// SIMATIC STEP 7 (V5.x) project Y_A start
// CPU: CPU 315
// station: Hardware
// station: SIMATIC 300(1)
// station: P_ADR_BUS
// program: S7 Program(3)

SYMBOL_TABLE
"Y_A"	FC 1	FC 1	// 星_三角 启动
"open"	I 0.0	BOOL	// 启动按钮
"stop"	I 0.1	BOOL	// 停止按钮
"over"	I 0.2	BOOL	// 过载保护
"T_km"	Q 4.0	BOOL	// 总接触器
"Y_km"	Q 4.1	BOOL	// 星点接触器
"A_km"	Q 4.2	BOOL	// 三角形接触器
"lamp"	Q 5.0	BOOL	// 运行指示灯
"timer0"	T 0	TIMER	// 星接延时
"timer1"	T 1	TIMER	// 断星接延时
"timer2"	T 2	TIMER	// 接通三角延时
END_SYMBOL_TABLE

FUNCTION "Y_A" : VOID	// FC 1
TITLE = 星_三角 启动电路
//这里星_三角 启动电路的功能模块。按启动按钮open后，运行指示lamp有指示，接触器T_km
//和Y_km接通，进行星形启动，时间为t0，然后断开T_km和Y_km，时间为t1，再接通A_km，延
//时t2时间后，再接通T_km，星三角启动完成。按停止按钮stop，或电路过载over，可停止电
//路运行。
VERSION : 0.1
VAR_INPUT
  open : BOOL ;	//启动按钮
  stop : BOOL ;	//停止按钮
  over : BOOL ;	//过载保护
  t0 : S5TIME ;	//星接延时时间
  t1 : S5TIME ;	//断开星接时间
  t2 : S5TIME ;	//接通三角时间
  timer0 : TIMER ;	//星接延时器
  timer1 : TIMER ;	//断星延时器
  timer2 : TIMER ;	//接角延时器
END_VAR
VAR_OUTPUT
  T_km : BOOL ;	//总接触器
  Y_km : BOOL ;	//星点接触器
  A_km : BOOL ;	//三角接触器
  lamp : BOOL ;	//运行指示
END_VAR
BEGIN
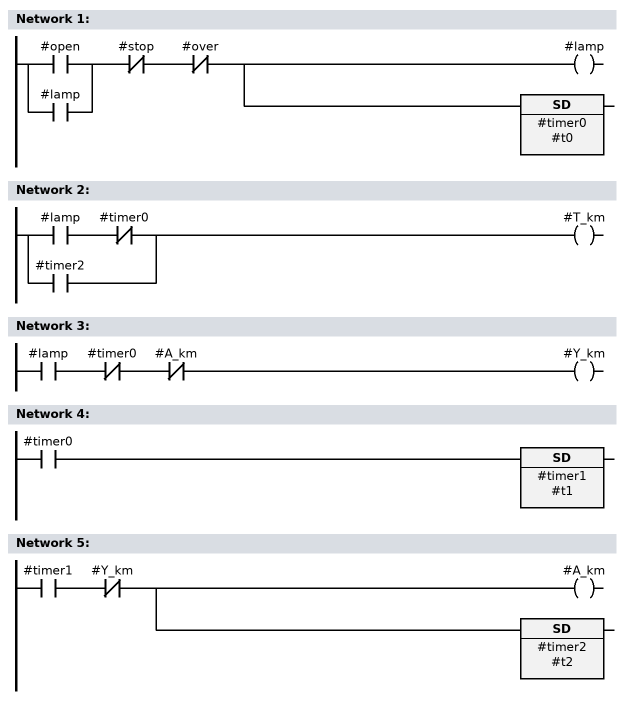
NETWORK
TITLE =
      A(;
      O     #open;
      O     #lamp;
      );
      AN    #stop;
      AN    #over;
      =     #lamp;
      L     #t0;
      SD    #timer0;
NETWORK
TITLE =
      A     #lamp;
      AN    #timer0;
      O     #timer2;
      =     #T_km;
NETWORK
TITLE =
      A     #lamp;
      AN    #timer0;
      AN    #A_km;
      =     #Y_km;
NETWORK
TITLE =
      A     #timer0;
      L     #t1;
      SD    #timer1;
NETWORK
TITLE =
      A     #timer1;
      AN    #Y_km;
      =     #A_km;
      L     #t2;
      SD    #timer2;
END_FUNCTION

ORGANIZATION_BLOCK OB 1
TITLE = "Main Program Sweep (Cycle)"
VERSION : 0.1
VAR_TEMP
  OB1_EV_CLASS : BYTE ;	//Bits 0-3 = 1 (Coming event), Bits 4-7 = 1 (Event class 1)
  OB1_SCAN_1 : BYTE ;	//1 (Cold restart scan 1 of OB 1), 3 (Scan 2-n of OB 1)
  OB1_PRIORITY : BYTE ;	//Priority of OB Execution
  OB1_OB_NUMBR : BYTE ;	//1 (Organization block 1, OB1)
  OB1_RESERVED_1 : BYTE ;	//Reserved for system
  OB1_RESERVED_2 : BYTE ;	//Reserved for system
  OB1_PREV_CYCLE : INT ;	//Cycle time of previous OB1 scan (milliseconds)
  OB1_MIN_CYCLE : INT ;	//Minimum cycle time of OB1 (milliseconds)
  OB1_MAX_CYCLE : INT ;	//Maximum cycle time of OB1 (milliseconds)
  OB1_DATE_TIME : DATE_AND_TIME ;	//Date and time OB1 started
END_VAR
BEGIN
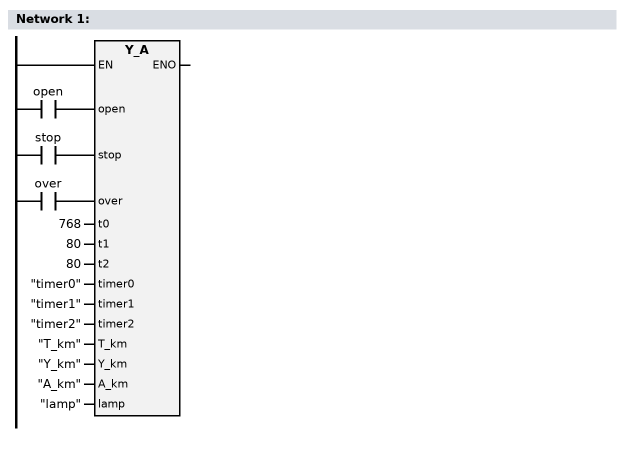
NETWORK
TITLE =
      A     "open";
      =     L 20.0;
      BLD   103;
      A     "stop";
      =     L 20.1;
      BLD   103;
      A     "over";
      =     L 20.2;
      BLD   103;
      CALL  "Y_A" (
           open                     := L 20.0,
           stop                     := L 20.1,
           over                     := L 20.2,
           t0                       := 768,
           t1                       := 80,
           t2                       := 80,
           timer0                   := "timer0",
           timer1                   := "timer1",
           timer2                   := "timer2",
           T_km                     := "T_km",
           Y_km                     := "Y_km",
           A_km                     := "A_km",
           lamp                     := "lamp");
      NOP   0;
END_ORGANIZATION_BLOCK
